FUNCTION_BLOCK Velocity_PI_REAL2 (* Composite Function Block Type *)
  (* Standard: 61499-2 *)
  (* Version 0.0, 2018-09-30, 4DIAC-IDE, 4DIAC-Consortium *)
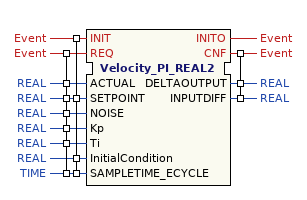
  EVENT_INPUT
    INIT WITH SETPOINT, InitialCondition, SAMPLETIME_ECYCLE; (* Initialization Request *)
    REQ WITH ACTUAL, NOISE, Kp, Ti, SETPOINT, SAMPLETIME_ECYCLE; (* Normal Execution Request *)
  END_EVENT
  EVENT_OUTPUT
    INITO; (* Initialization Confirm *)
    CNF WITH DELTAOUTPUT, INPUTDIFF; (* Execution Confirmation *)
  END_EVENT
  VAR_INPUT
    ACTUAL : REAL;
    SETPOINT : REAL;
    NOISE : REAL;
    Kp : REAL;
    Ti : REAL;
    InitialCondition : REAL;
    SAMPLETIME_ECYCLE : TIME;
  END_VAR
  VAR_OUTPUT
    DELTAOUTPUT : REAL;
    INPUTDIFF : REAL;
  END_VAR
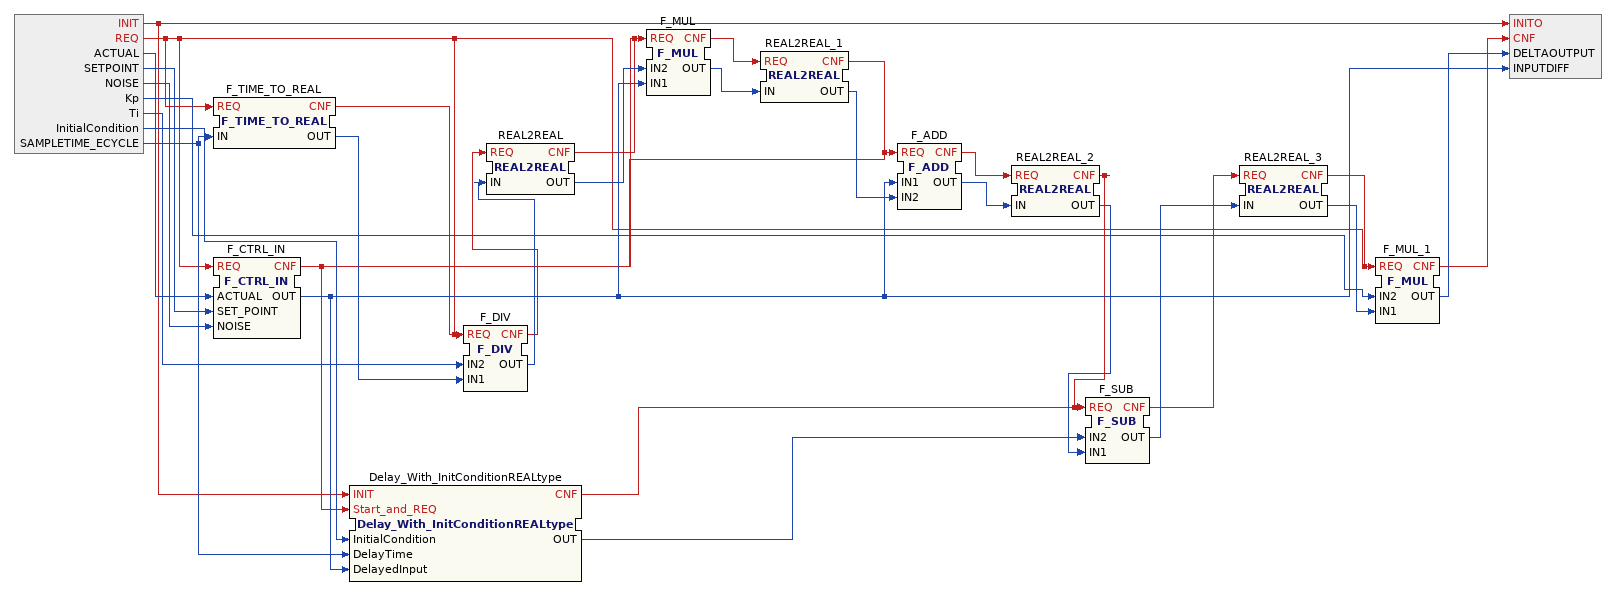
  FBS
    F_CTRL_IN : F_CTRL_IN;
    F_TIME_TO_REAL : F_TIME_TO_REAL;
    Delay_With_InitConditionREALtype : Delay_With_InitConditionREALtype;
    F_DIV : F_DIV;
    REAL2REAL : REAL2REAL;
    F_MUL : F_MUL;
    REAL2REAL_1 : REAL2REAL;
    F_ADD : F_ADD;
    REAL2REAL_2 : REAL2REAL;
    F_SUB : F_SUB;
    REAL2REAL_3 : REAL2REAL;
    F_MUL_1 : F_MUL;
  END_FBS
  EVENT_CONNECTIONS
    INIT TO Delay_With_InitConditionREALtype.INIT;
    REQ TO F_TIME_TO_REAL.REQ;
    INIT TO INITO;
    REQ TO F_CTRL_IN.REQ;
    REQ TO F_MUL_1.REQ;
    F_CTRL_IN.CNF TO Delay_With_InitConditionREALtype.Start_and_REQ;
    Delay_With_InitConditionREALtype.CNF TO F_SUB.REQ;
    F_SUB.CNF TO REAL2REAL_3.REQ;
    REAL2REAL_3.CNF TO F_MUL_1.REQ;
    REQ TO F_DIV.REQ;
    F_TIME_TO_REAL.CNF TO F_DIV.REQ;
    F_DIV.CNF TO REAL2REAL.REQ;
    REAL2REAL.CNF TO F_MUL.REQ;
    F_CTRL_IN.CNF TO F_MUL.REQ;
    F_MUL.CNF TO REAL2REAL_1.REQ;
    F_CTRL_IN.CNF TO F_ADD.REQ;
    REAL2REAL_1.CNF TO F_ADD.REQ;
    F_ADD.CNF TO REAL2REAL_2.REQ;
    REAL2REAL_2.CNF TO F_SUB.REQ;
    F_MUL_1.CNF TO CNF;
  END_CONNECTIONS
  DATA_CONNECTIONS
    SAMPLETIME_ECYCLE TO F_TIME_TO_REAL.IN;
    ACTUAL TO F_CTRL_IN.ACTUAL;
    SETPOINT TO F_CTRL_IN.SET_POINT;
    NOISE TO F_CTRL_IN.NOISE;
    Kp TO F_MUL_1.IN2;
    InitialCondition TO Delay_With_InitConditionREALtype.InitialCondition;
    SAMPLETIME_ECYCLE TO Delay_With_InitConditionREALtype.DelayTime;
    F_CTRL_IN.OUT TO Delay_With_InitConditionREALtype.DelayedInput;
    Delay_With_InitConditionREALtype.OUT TO F_SUB.IN2;
    F_SUB.OUT TO REAL2REAL_3.IN;
    REAL2REAL_3.OUT TO F_MUL_1.IN1;
    Ti TO F_DIV.IN2;
    F_TIME_TO_REAL.OUT TO F_DIV.IN1;
    F_DIV.OUT TO REAL2REAL.IN;
    REAL2REAL.OUT TO F_MUL.IN2;
    F_CTRL_IN.OUT TO F_MUL.IN1;
    F_CTRL_IN.OUT TO INPUTDIFF;
    F_CTRL_IN.OUT TO F_ADD.IN1;
    F_MUL.OUT TO REAL2REAL_1.IN;
    REAL2REAL_1.OUT TO F_ADD.IN2;
    F_ADD.OUT TO REAL2REAL_2.IN;
    REAL2REAL_2.OUT TO F_SUB.IN1;
    F_MUL_1.OUT TO DELTAOUTPUT;
  END_CONNECTIONS
END_FUNCTION_BLOCK
